PROGRAM PRG_Fault_SMAC
VAR
	i					: INT;
	bTest				: BOOL;
END_VAR
VAR_IN_OUT
  aAlarms  : ARRAY[0..3] OF ST_Events;
END_VAR

IF GVL_PERSISTENT.bSMACEnable THEN 
ACT_FaultTrig();
END_IF

(************************************** Faults reset **********************************************)
IF   bResetButtonRisingEdge THEN 
	FOR i := 0 TO 127 DO
		GVL_MASTER.stAlarms[3].aEventFlags[i] := FALSE;
	END_FOR
END_IF
//===============================================================
//Initialize event texts on first scan
IF NOT GVL_MASTER.stAlarms[3].bEventTextsSet THEN
	SetEventTexts();
	GVL_MASTER.stAlarms[3].bEventTextsSet := TRUE;
END_IF


(***************************************************************************************************)
//Immediate fault
GVL_MASTER.stAlarms[3].bImmediateFault := FALSE;
FOR i := 0 TO 32DO
	GVL_MASTER.stAlarms[3].bImmediateFault := GVL_MASTER.stAlarms[3].bImmediateFault OR GVL_MASTER.stAlarms[3].aEventFlags[i];
END_FOR

//Cycle stop fault
GVL_MASTER.stAlarms[3].bCycleStopFault := FALSE;
FOR i := 33 TO 79 DO
	GVL_MASTER.stAlarms[3].bCycleStopFault := GVL_MASTER.stAlarms[3].bCycleStopFault OR GVL_MASTER.stAlarms[3].aEventFlags[i];
END_FOR

//Cycle stop REQUEST
GVL_MASTER.stAlarms[3].bCycleStopRequest := FALSE;
FOR i := 80 TO 99 DO
	GVL_MASTER.stAlarms[3].bCycleStopRequest := GVL_MASTER.stAlarms[3].bCycleStopRequest OR GVL_MASTER.stAlarms[3].aEventFlags[i];
END_FOR

ACTION ACT_FaultTrig:

//Station 3 - SMAC Linear Servo error
IF stSmacIO.inStatusWordLinear.13 THEN 
	stAlarms[3].aEventFlags[2] := TRUE;
	bTest							:= TRUE;
END_IF
//Station 3 - SMAC Rotative Servo error
IF stSmacIO.inStatusWordRotative.13 THEN 
	stAlarms[3].aEventFlags[4] := TRUE;
	bTest							:= TRUE;
END_IF
//Station 3 - SMAC STO Fault
IF stSmacIO.inStatusWordRotative.15 OR stSmacIO.inStatusWordLinear.15 THEN 
	stAlarms[3].aEventFlags[5] := TRUE;
	bTest							:= TRUE;
END_IF
//Station 3 - SMAC I2T Fault
IF stSmacIO.inStatusWordRotative.18 OR stSmacIO.inStatusWordLinear.18 THEN 
	stAlarms[3].aEventFlags[6] := TRUE;
	bTest							:= TRUE;
END_IF
//Station 3 - SMAC Over temperature Fault
IF stSmacIO.inStatusWordRotative.19 OR stSmacIO.inStatusWordLinear.19 THEN 
	stAlarms[3].aEventFlags[7] := TRUE;
	bTest							:= TRUE;
END_IF




//Station 3 - SMAC Homing Time Out
GVL_MASTER.stAlarms[3].aEventTimers[80]
(IN := (S_Master_SMAC.eState = E_SmacState.HOMING),PT:= T#30S );
IF GVL_MASTER.stAlarms[3].aEventTimers[80].Q  THEN 
	GVL_MASTER.stAlarms[3].aEventFlags[80] := TRUE;
END_IF
//Station 3 - SMAC Linear Homing fail
GVL_MASTER.stAlarms[3].aEventTimers[81]
(IN := (S_Master_SMAC.eState = E_SmacState.HOMING) AND stSmacIO.inStatusWordLinear.7 ,PT:= T#20S );
IF GVL_MASTER.stAlarms[3].aEventTimers[81].Q THEN 
	stAlarms[3].aEventFlags[81] := TRUE;
END_IF
//Station 3 - SMAC Linear Phasing fail
GVL_MASTER.stAlarms[3].aEventTimers[82]
(IN := (S_Master_SMAC.eState = E_SmacState.HOMING) AND stSmacIO.inStatusWordLinear.9 ,PT:= T#20S );
IF GVL_MASTER.stAlarms[3].aEventTimers[82].Q THEN
	stAlarms[3].aEventFlags[82] := TRUE;
END_IF
//Station 3 - SMAC Rotative Homing fail
GVL_MASTER.stAlarms[3].aEventTimers[83]
(IN := (S_Master_SMAC.eState = E_SmacState.HOMING) AND stSmacIO.inStatusWordRotative.7 ,PT:= T#20S );
IF GVL_MASTER.stAlarms[3].aEventTimers[83].Q THEN 
	stAlarms[3].aEventFlags[83] := TRUE;
END_IF
//Station 3 - SMAC Rotative Phasing fail
GVL_MASTER.stAlarms[3].aEventTimers[84]
(IN := (S_Master_SMAC.eState = E_SmacState.HOMING) AND stSmacIO.inStatusWordRotative.9 ,PT:= T#20S );
IF GVL_MASTER.stAlarms[3].aEventTimers[84].Q THEN 
	stAlarms[3].aEventFlags[84] := TRUE;
END_IF
END_ACTION

METHOD SetEventTexts : BOOL
VAR_INPUT
END_VAR
//Immediate Faults
GVL_MASTER.stAlarms[3].aEventTexts[1] := 'Station 3 - SMAC Linear General Fault';
GVL_MASTER.stAlarms[3].aEventTexts[2] := 'Station 3 - SMAC Linear Servo error';
GVL_MASTER.stAlarms[3].aEventTexts[3] := 'Station 3 - SMAC Rotative General Fault';
GVL_MASTER.stAlarms[3].aEventTexts[4] := 'Station 3 - SMAC Rotative Servo error';
GVL_MASTER.stAlarms[3].aEventTexts[5] := 'Station 3 - SMAC STO Fault';
GVL_MASTER.stAlarms[3].aEventTexts[6] := 'Station 3 - SMAC I2T Fault';
GVL_MASTER.stAlarms[3].aEventTexts[7] := 'Station 3 - SMAC Over temperature Fault';
GVL_MASTER.stAlarms[3].aEventTexts[8] := '';
GVL_MASTER.stAlarms[3].aEventTexts[9] := ''; 
GVL_MASTER.stAlarms[3].aEventTexts[10] := ''; 
GVL_MASTER.stAlarms[3].aEventTexts[11] := '';
GVL_MASTER.stAlarms[3].aEventTexts[12] := '';
GVL_MASTER.stAlarms[3].aEventTexts[13] := '';
GVL_MASTER.stAlarms[3].aEventTexts[14] := '';
GVL_MASTER.stAlarms[3].aEventTexts[15] := '';
GVL_MASTER.stAlarms[3].aEventTexts[16] := '';
GVL_MASTER.stAlarms[3].aEventTexts[17] := '';
GVL_MASTER.stAlarms[3].aEventTexts[18] := '';
GVL_MASTER.stAlarms[3].aEventTexts[19] := '';
GVL_MASTER.stAlarms[3].aEventTexts[20] := '';
GVL_MASTER.stAlarms[3].aEventTexts[21] := '';
GVL_MASTER.stAlarms[3].aEventTexts[22] := '';
GVL_MASTER.stAlarms[3].aEventTexts[28] := '';
GVL_MASTER.stAlarms[3].aEventTexts[29] := '';
GVL_MASTER.stAlarms[3].aEventTexts[30] := '';

//Cycle Stop Requests

GVL_MASTER.stAlarms[3].aEventTexts[80] := 'Station 3 - SMAC Homing Time Out';
GVL_MASTER.stAlarms[3].aEventTexts[81] := 'Station 3 - SMAC Linear Homing fail';
GVL_MASTER.stAlarms[3].aEventTexts[82] := 'Station 3 - SMAC Linear Phasing fail';
GVL_MASTER.stAlarms[3].aEventTexts[84] := 'Station 3 - SMAC Rotative Homing fail';
GVL_MASTER.stAlarms[3].aEventTexts[85] := 'Station 3 - SMAC Rotative Phasing fail';
GVL_MASTER.stAlarms[3].aEventTexts[86] := '';
GVL_MASTER.stAlarms[3].aEventTexts[87] := ''; 
GVL_MASTER.stAlarms[3].aEventTexts[88] := '';
GVL_MASTER.stAlarms[3].aEventTexts[89] := '';
END_METHOD

END_PROGRAM

(* stored: Version 1.1.0.1, ProductVersion 3.1.4024.12
   POU PRG_Fault_SMAC: Id {555cc3af-ba28-485f-a0a0-3fcc4c7f4d43}, SpecialFunc None
   Action ACT_FaultTrig: Id {5ced6ccf-eb80-4f52-980a-c990eb91b259}
   Method SetEventTexts: Id {440556e1-2869-4fbc-8381-5109ef053a3c} *)
